# EPICS substitutions: TPG300/TPG300-IOC-01App/Db/TPG300_channels.substitutions
file kynctm3k.template {

pattern {PORT, P, CHAN, IFTEST}
{"\$(PORT)", "\$(P)", "A1", "\$(IFPRESSURA1)"}
{"\$(PORT)", "\$(P)", "A2", "\$(IFPRESSURA2)"}
{"\$(PORT)", "\$(P)", "B1", "\$(IFPRESSURB1)"}
{"\$(PORT)", "\$(P)", "B2", "\$(IFPRESSURB2)"}

}
